FUNCTION_BLOCK INTERNAL FB_CylinderTestAlternative
VAR
	fbCylinder : FB_CylinderAlternative;
END_VAR

{attribute 'TcRpcEnable'}
METHOD MoveCylinderToHome : BOOL
MoveCylinderToHome := fbCylinder.MoveToHome();
END_METHOD

{attribute 'TcRpcEnable'}
METHOD MoveCylinderToWork : BOOL
MoveCylinderToWork := fbCylinder.MoveToWork();
END_METHOD

END_FUNCTION_BLOCK

(* stored: Version 1.1.0.1, ProductVersion 3.1.4024.4
   POU FB_CylinderTestAlternative: Id {721255ca-134a-4131-8eee-ee5e15e5be2f}, SpecialFunc None
   Method MoveCylinderToHome: Id {3a42f3af-fba8-4502-bcfe-dbc0031d9218}
   Method MoveCylinderToWork: Id {5e3db9ed-2149-436d-bf64-583f9bd6bf1d} *)
